PROGRAM FilterWheelControl
VAR_INPUT
	// enable the axis
	Enable:				BOOL;
	// reset the axis(-error)
	Reset:				BOOL;
	// move counter-clockwise
	left:				BOOL;
	// move clockwise
	right:				BOOL;
	// TRUE, if the filter is in position and wheel has come to rest
	Ready:				BOOL;
	// filter position
	filter_position: 	USINT;
	// move to given position
	MoveAxis: 			BOOL;
	// calibrate the axis
	HomeAxis:			BOOL;
END_VAR
VAR_OUTPUT
	// is true if an error occurred
	error: 				BOOL;
	// number of current axis error
	ErrorID:			UDINT;
	act_position:		LREAL;
	// axis has been calibrated
	Calibrated :		BOOL;
END_VAR
VAR
	FilterWheelAxis:	FB_Axis2;
	// axis position to set to with `MoveAxis`
	position:			LREAL;
	// current filter determined from the axis position
	actual_filter:		USINT;
	FilterWheelEvent:	FB_EventLog;
	CalibratedEvent:	FB_EventLog;
	FilterReadyEvent:	FB_Eventlog;
	// last known filter position
	last_filter_position:	USINT;
END_VAR
VAR CONSTANT
	// total number of filters in the filter wheel
	filters:			USINT := 24;
	// current position of the calibration cam. Apply an offset here if necessary
	calibration_position:	LREAL := 0.0;
END_VAR

(* This program controls the filter wheel. 
The current optical filter is selected through `filter_position`.
The number of filters is hard coded to 24.

*)

// limit desired filter_position to [0...filters-1]
filter_position := filter_position MOD filters;
// calculate the actual filter position
actual_filter := LREAL_TO_USINT((360.0 - act_position) * filters / 360.0) MOD filters;

Ready := (filter_position = actual_filter) AND FilterWheelAxis.Standstill;

// TODO: Enable only on filter change
IF Enable THEN
	IF FilterWheelAxis.Calibrated THEN
		HomeAxis := FALSE;
		// if we are on automatic mode then position the filterwheel
		position := MODABS(360.0 - 360.0 * WORD_TO_LREAL(filter_position) / WORD_TO_LREAL(filters), 360.0);
		MoveAxis := filter_position <> actual_filter AND FilterWheelAxis.Standstill;
	ELSE
		position := calibration_position;
		IF FilterWheelAxis.Ready THEN
			HomeAxis := TRUE;
		END_IF
	END_IF
END_IF

Calibrated := FilterWheelAxis.Calibrated;

FilterWheelAxis(
	Enable := 			Enable,
	Reset := 			Reset,
	MoveAxis :=			MoveAxis,
	HomeAxis :=			HomeAxis,
	HomingMode :=		MC_ForceCalibration,
	Position := 		position, 
	Velocity :=			60.0,
	Enable_Positive :=  TRUE,
	Enable_Negative := 	TRUE,
	Jog_Forward :=		left,
	Jog_Backwards := 	right,
	bCalibrationCam :=	NOT GVL_FilterWheel.bCalibrationCam,
	isModuloAxis :=		TRUE,
	ActualPosition => 	act_position,
	Error => 			error,
	ErrorID => 			ErrorID,
	AxisRef :=			GVL_FilterWheel.FilterWheel_AxisRef);

IF FilterWheelAxis.MoveDone THEN
	MoveAxis := FALSE;
END_IF

IF FilterWheelAxis.HomeDone THEN
	HomeAxis := FALSE;
END_IF
	
IF FilterWheelAxis.ResetDone THEN
	reset := FALSE;
END_IF

IF actual_filter <> last_filter_position THEN
	MAIN.MQTTClient.Publish('telescope', 'dome', 'FilterPosition', WORD_TO_STRING(actual_filter));
	last_filter_position := actual_filter;
END_IF

FilterWheelEvent(	
	Trigger := 		Error, 
	Level := 		ADSLOG_MSGTYPE_ERROR,
	FormatString :=	'Filter Wheel Axis Error: %s',
	OnMessage := 	NCError_TO_STRING(ErrorID),
	OffMEssage := 	'OK',
	OffLevel := 	ADSLOG_MSGTYPE_HINT);
	
CalibratedEvent(
	Trigger :=		Calibrated,
	Level := 		ADSLOG_MSGTYPE_HINT,
	FormatString :=	'%s',
	OnMessage := 	'Filter wheel is calibrated.');
	
FilterReadyEvent(
	Trigger :=		(filter_position = actual_filter) AND Calibrated,
	Level := 		ADSLOG_MSGTYPE_HINT,
	FormatString :=	'Filter position %s is ready.',
	OnMessage := 	WORD_TO_STRING(actual_filter));

END_PROGRAM

(* stored: Version 1.1.0.1, ProductVersion 3.1.4024.9
   POU FilterWheelControl: Id {f0e4f375-0934-4386-a9fa-94537c34c7e1}, SpecialFunc None *)
